	n_CP1_max_speed := GVL_RESD.n_Concrete_Pump_Max_Speed,
	n_CP1_target_speed := UINT_TO_INT(GVL_ROB.in_CP1_set_speed),

	// Admixture pump (High)
	b_AP1_Power_On := GVL_ROB.ib_AP1_power_on,
	b_AP1_Run := GVL_ROB.ib_AP1_set_run,
	b_AP1_Flush_On := GVL_ROB.ib_AP1_flush_on,
	b_AP1_Check_On := GVL_ROB.ib_AP1_check_on,
	
	n_AP1_Flowrate_mode := TRUE,
	n_AP1_Max_Flowrate := UINT_TO_INT(GVL_ROB.on_AP1_max_flowrate),
	n_AP1_Operate_Flowrate := REAL_TO_UDINT((UINT_TO_REAL(GVL_ROB.in_AP1_set_flowrate*10))),
	n_AP1_Check_Flowrate := REAL_TO_UDINT((UINT_TO_REAL(GVL_ROB.in_AP1_set_check_flowrate*10))),
	n_AP1_Flush_Flowrate := REAL_TO_UDINT((UINT_TO_REAL(GVL_ROB.in_AP1_set_flush_flowrate*10))),
	n_AP1_Dosing_factor := UINT_TO_INT(GVL_ROB.in_AP1_set_dosing_factor),
	
	// Admixture pump (High)
	b_SP1_Power_On := GVL_ROB.ib_SP1_power_on,
	b_SP1_Run := GVL_ROB.ib_SP1_set_run,
	b_SP1_Flush_On := GVL_ROB.ib_SP1_flush_on,
	b_SP1_Check_On := GVL_ROB.ib_SP1_set_check_on,
	
	n_SP1_Flowrate_mode := TRUE,
	n_SP1_Max_Flowrate := UINT_TO_INT(GVL_ROB.on_SP1_max_flowrate),
	n_SP1_Operate_Flowrate := REAL_TO_UDINT((UINT_TO_REAL(GVL_ROB.in_SP1_set_flowrate*10))),
	n_SP1_Check_Flowrate := REAL_TO_UDINT((UINT_TO_REAL(GVL_ROB.in_SP1_set_check_flowrate*10))),
	n_SP1_Flush_Flowrate := REAL_TO_UDINT((UINT_TO_REAL(GVL_ROB.in_SP1_flush_flowrate*10))),
	n_SP1_Dosing_factor := UINT_TO_INT(GVL_ROB.in_SP1_dosing_factor),
	);

//***********************************************************************************
// Inline Mixer
//***********************************************************************************
	//mixer 
Mixer1_2(
	Mixer1			:= GVL.Axis_Mixer1,
	Mixer2			:= GVL.Axis_Mixer2,
	f_Velocity		:= GVL.f_MI1_MaxSpeed,
	b_JogForward	:= FALSE,
	b_JogBackwards	:= fb_SetOutputDataToIO.b_MI1_set_run,
	b_Enable		:= fb_SetOutputDataToIO.b_Ml1_Enable AND GVL_IO.ib_CC1_Safety_Ready,
	b_Reset			:= GVL_ROB.ib_CC1_reset OR GVL_IO.ib_CC1_Button_Reset,
	f_Override		:= GVL.n_MI1_OverrideSpeed,
	);
	(*
	fb_MC_SetPosition(
	Axis			:= GVL.Axis_Mixer2,
	memory			:= 1,
	Feedback		:= 0);*)
pos:=GVL.Axis_Mixer2.NcToPlc.ModuloActPos;
GVL.b_MI1_ReadToDrive:=Mixer1_2.b_ReadyToDrive;
P_MI1_OnOff(b_set_run := fb_SetOutputDataToIO.b_MI1_set_run,);

//***********************************************************************************
// Concrete Pump
//***********************************************************************************

// concrete pump power control is from pump itself
P_CP1_Enable();
P_CP1_Check(b_set_run := fb_SetOutputDataToIO.b_CP1_Forward_On,
			b_check_mode_on := fb_SetOutputDataToIO.b_CP1_Check_On,
			t_check_duration := fb_setConfig._t_CP1_Check_Duration,
			);


//***********************************************************************************
// Acceleration Pump
//***********************************************************************************

// Acceleration Pump 1 check
P_AP1_Check(b_set_run := fb_SetOutputDataToIO.b_AP1_Run,
			b_check_mode_on := fb_SetOutputDataToIO.b_AP1_Check_On,
			t_check_duration := fb_setConfig._t_AP1_Check_Duration,
			);
// Check for Acceleration Pump 1 state
IF NOT fb_SetOutputDataToIO.b_AP1_Check_On THEN
//
// Acceleration Pump 1 On/Off
	P_AP1_OnOff(b_set_run := fb_SetOutputDataToIO.b_AP1_Run);
END_IF

//***********************************************************************************
// Superplasticizer Pump
//***********************************************************************************

// Superplasticizer Pump 1 Check (220916 WT
P_SP1_Check(b_set_run := fb_SetOutputDataToIO.b_SP1_Run,
			b_check_mode_on := fb_SetOutputDataToIO.b_SP1_Check_On,
			t_check_duration := fb_setConfig._t_SP1_Check_Duration,
			);
IF NOT fb_SetOutputDataToIO.b_SP1_Check_On THEN
	P_SP1_OnOff(b_set_run := fb_SetOutputDataToIO.b_SP1_Run);
END_IF

//***********************************************************************************
// Get out put data from PLC
//***********************************************************************************
fb_getOutputData(
	
	//CC1
	b_mode_manual := GVL_ROB.ob_mode_manual,
	b_mode_laptop := GVL_ROB.ob_mode_laptop, 	
	b_mode_robot := GVL_ROB.ob_mode_robot, 
	b_CC1_power_on := GVL_ROB.ob_CC1_power_on, 
	n_current_mode := GVL_ROB.on_current_mode,

	//MI1
	b_MI1_Is_Run := GVL_ROB.ob_MI1_is_run,
	b_MI1_is_ready := GVL_ROB.ob_MI1_is_ready,
	n_MI1_status_SpeedM1 := GVL_ROB.on_MI1_status_speed_motor_1,
	n_MI1_status_SpeedM2 := GVL_ROB.on_MI1_status_speed_motor_2,
	f_Status_Torque_Motor_1 := GVL_ROB.on_MI1_status_torque_motor_1,
	f_Status_Torque_Motor_2 := GVL_ROB.on_MI1_status_torque_motor_2,
	f_MI1_status_temperature_funnel_outlet := GVL_ROB.on_MI1_status_temperature_funnel_outlet,
	f_MI1_status_Pressure_funnel_inlet := GVL_ROB.on_MI1_status_pressure_funnel_inlet, 	
	f_MI1_status_temperature_motor_1  := GVL_ROB.on_MI1_status_temperature_motor_1, 			 
	f_MI1_status_temperature_motor_2  := GVL_ROB.on_MI1_status_temperature_motor_2,

	//CP1
	b_CP1_is_run := GVL_ROB.ob_CP1_is_run,
	b_CP1_is_ready := GVL_ROB.ob_CP1_is_ready,
	b_CP1_power_on := GVL_ROB.ob_CP1_power_on,
	b_CP1_safety_grid_on := GVL_ROB.ob_CP1_safety_grid_on,
	b_CP1_drive_error := GVL_ROB.ob_CP1_drive_error,
	
	f_CP1_status_temperature_concrete_fresh := GVL_ROB.on_CP1_status_temperature_concrete_fresh,
	f_CP1_status_temperature_Concrete_pump := GVL_ROB.on_CP1_status_temperature_concrete_pump,
	f_CP1_status_pressure_Concrete_pump := GVL_ROB.on_CP1_status_pressure_concrete_pump,
	
	//AP1
	b_AP1_is_run := GVL_ROB.ob_AP1_is_run,
	b_AP1_is_ready := GVL_ROB.ob_AP1_is_ready,
	b_AP1_no_error := GVL_ROB.ob_AP1_no_error,
	
	//SP1
	b_SP1_is_run := GVL_ROB.ob_SP1_is_run,
	b_SP1_is_ready := GVL_ROB.ob_SP1_is_ready,
	b_SP1_no_error := GVL_ROB.ob_SP1_no_error,
);

END_PROGRAM

// ---- POUs/temp.TcPOU
PROGRAM temp
VAR
END_VAR

(*
// Concrete pump (CP1) *****
	// Digital output from robot (mapping from 16 to 23 in robotstudio )
		arr_CP1_DOSlot := F_CONVERT_BYTE_TO_BIT(GVL_PN.DO_From_ROB[2]);
		GVL_ROB.ib_CP1_forward_on := arr_CP1_DOSlot[0]; // #16
		GVL_ROB.ib_CP1_backward_on := arr_CP1_DOSlot[1];		// 241219 Backward is not working from the conctroller
		GVL_ROB.ib_CP1_check_on := arr_CP1_DOSlot[2];
		GVL_ROB.ib_CP1_flush_on := arr_CP1_DOSlot[3];

	// Group output from Robot ( mapping from 62 to 76, 8*2Bytes in robotstudio)
		F_Convert_2Byte_to_Int(GVL_ROB.in_CP1_set_speed, arr_GOSlot[62], arr_GOSlot[63]); // 0 to 75 [rpm] #62
		F_Convert_2Byte_to_Int(GVL_ROB.in_CP1_set_flowrate, arr_GOSlot[64], arr_GOSlot[65]); // 0 to 16 [l/min]
		F_Convert_2Byte_to_Int(GVL_ROB.in_CP1_set_dosing_volume, arr_GOSlot[66], arr_GOSlot[67]); // calibration in 230926 WT 0.32
		F_Convert_2Byte_to_Int(GVL_ROB.in_CP1_set_check_Flowrate, arr_GOSlot[68], arr_GOSlot[69]);	// [l/min]
		F_Convert_2Byte_to_Int(GVL_ROB.in_CP1_concrete_density, arr_GOSlot[70], arr_GOSlot[71]); // [g/ml]
		F_Convert_2Byte_to_Int(GVL_ROB.in_CP1_concrete_mass, arr_GOSlot[72], arr_GOSlot[73]); // [g]
		F_Convert_2Byte_to_Int(GVL_ROB.in_CP1_set_flush_flowrate, arr_GOSlot[74], arr_GOSlot[75]); // [l/min]
		// F_Convert_2Byte_to_Int(GVL_ROB.t_CP1_set_check_duration, arr_GOSlot[76], arr_GOSlot[77]);	 check with 32 bit


	// Digital input to robot (mapping from 16 to 23 in robotstudio)
		//arr_CP1_DISlot := F_CONVERT_BYTE_TO_BIT(GVL_PN.DI_To_ROB[2]);
		arr_CP1_DISlot[0] := GVL_ROB.ob_CP1_is_run; // #16
		arr_CP1_DISlot[1] := GVL_ROB.ob_CP1_is_ready;

	// Group Input To Robot (mapping from 77 to 91, 8*2Bytes in robotstudio)
		F_Convert_Int_to_2Byte(GVL_ROB.on_CP1_status_temperature_concrete_fresh, arr_GISlot[77], arr_GISlot[78]); // [°C]
		F_Convert_Int_to_2Byte(GVL_ROB.on_CP1_status_temperature_Concrete_pump, arr_GISlot[79], arr_GISlot[80]); // [°C]
		F_Convert_Int_to_2Byte(GVL_ROB.on_CP1_status_pressure_Concrete_pump, arr_GISlot[81], arr_GISlot[82]); // [ bar]




// Admixture pump, High dosage ViscoTech Pump *****
	// Digital output from robot (mapping from 24 to 31 in robotstudio )
		arr_AP1_DOSlot := F_CONVERT_BYTE_TO_BIT(GVL_PN.DO_From_ROB[3]);
		GVL_ROB.ib_AP1_set_run := arr_AP1_DOSlot[0]; // #24
		GVL_ROB.ib_AP1_check_on := arr_AP1_DOSlot[1];
		GVL_ROB.ib_AP1_flush_on := arr_AP1_DOSlot[2];

	// Group output from Robot ( mapping from 77 to 91, 8*2Bytes in robotstudio)
		F_Convert_2Byte_to_Int(GVL_ROB.in_AP1_set_flowrate, arr_GOSlot[77], arr_GOSlot[78]); // **** [ml/min] #77
		F_Convert_2Byte_to_Int(GVL_ROB.in_AP1_set_dosing_factor, arr_GOSlot[79], arr_GOSlot[80]);
		F_Convert_2Byte_to_Int(GVL_ROB.in_AP1_set_check_flowrate, arr_GOSlot[81], arr_GOSlot[82]);
		F_Convert_2Byte_to_Int(GVL_ROB.in_AP1_material_density, arr_GOSlot[83], arr_GOSlot[84]);
		F_Convert_2Byte_to_Int(GVL_ROB.in_AP1_material_mass, arr_GOSlot[85], arr_GOSlot[86]);

		F_Convert_2Byte_to_Int(GVL_ROB.in_AP1_set_dosing_factor, arr_GOSlot[79], arr_GOSlot[80]);
		F_Convert_2Byte_to_Int(GVL_ROB.in_AP1_flush_flowrate, arr_GOSlot[81], arr_GOSlot[82]);
		// F_Convert_2Byte_to_Int(GVL_ROB.t_AP1_set_check_duration, arr_GOSlot[83], arr_GOSlot[84]); check with 32 bit

	// Digital input to robot (mapping from 24 to 31 in robotstudio)
		//arr_AP1_DISlot := F_CONVERT_BYTE_TO_BIT(GVL_PN.DI_To_ROB[3]);	// #24
		arr_AP1_DISlot[0] := GVL_ROB.ob_AP1_is_run;

	// Group Input To Robot (mapping from 92 to 106, 8*2Bytes in robotstudio)
		F_Convert_2Byte_to_Int(GVL_ROB.on_AP1_max_flowrate, arr_GOSlot[92], arr_GOSlot[93]); // [l/min]



// Admixture pump, Low dosage ViscoTech Pump *****
	// Digital output from robot (mapping from 32 to 39 in robotstudio )
		//arr_SP1_DOSlot := F_CONVERT_BYTE_TO_BIT(GVL_PN.DO_From_ROB[4]);
		GVL_ROB.ib_SP1_set_run := arr_SP1_DOSlot[0]; // #32
		GVL_ROB.ib_SP1_set_check_on := arr_SP1_DOSlot[1];
		GVL_ROB.ib_SP1_flush_on := arr_SP1_DOSlot[2];

	// Group output from Robot ( mapping from 92 to 106, 8*2Bytes in robotstudio)
		F_Convert_2Byte_to_Int(GVL_ROB.in_SP1_set_flowrate, arr_GOSlot[92], arr_GOSlot[93]); // **** [ml/min] #92
		F_Convert_2Byte_to_Int(GVL_ROB.in_SP1_dosing_factor, arr_GOSlot[93], arr_GOSlot[94]);
		F_Convert_2Byte_to_Int(GVL_ROB.in_SP1_set_check_flowrate, arr_GOSlot[95], arr_GOSlot[96]);
		F_Convert_2Byte_to_Int(GVL_ROB.in_SP1_material_density, arr_GOSlot[97], arr_GOSlot[98]);
		F_Convert_2Byte_to_Int(GVL_ROB.in_SP1_material_mass, arr_GOSlot[99], arr_GOSlot[100]);
		F_Convert_2Byte_to_Int(GVL_ROB.in_SP1_flush_flowrate, arr_GOSlot[101], arr_GOSlot[102]);
		// F_Convert_2Byte_to_Int(GVL_ROB.t_SP1_Check_Duration, arr_GOSlot[103], arr_GOSlot[104]); // Check with 32 bit

	// Digital input to robot (mapping from 32 to 39 in robotstudio)
		//arr_SP1_DISlot := F_CONVERT_BYTE_TO_BIT(GVL_PN.DI_To_ROB[4]);
		GVL_ROB.ob_SP1_is_run := arr_SP1_DISlot[0]; // #32

	// Group Input To Robot (mapping from 106 to 120, 8*2Bytes in robotstudio)
		F_Convert_2Byte_to_Int(GVL_ROB.on_SP1_max_flowrate, arr_GOSlot[106], arr_GOSlot[107]); // [l/min]>



// Spare Component *****
	// Digital output from robot (mapping from 40 to .. in robotstudio )
		// Template
		// arr_SP1_DOSlot := F_Convert_Byte_to_Bit(GVL_PN.DO_From_ROB[4]);
		// GVL_ROB.ib_SP1_set_run := arr_SP1_DOSlot[0];

	// Group output from Robot ( mapping from 107 to .., 8*2Bytes in robotstudio)
		// F_Convert_2Byte_to_Int(GVL_ROB.in_SP1_set_flowrate, arr_GOSlot[92], arr_GOSlot[93]);
	// Digital input to robot (mapping from 40 to .. in robotstudio)
		// Template
		// arr_SP1_DISlot := F_Convert_Byte_to_Bit(GVL_PN.DI_To_ROB[4]);
		// GVL_ROB.ob_SP1_is_run:= arr_SP1_DISlot[0]; // #32

	// Group Input To Robot (mapping from 121 to .., 8*2Bytes in robotstudio)
		// F_Convert_2Byte_to_Int(GVL_ROB.on_SP1_max_flowrate, arr_GOSlot[106], arr_GOSlot[107]);
//
*)

END_PROGRAM

// ---- POUs/Utils/F_Convert_2Byte_to_Real.TcPOU
FUNCTION F_Convert_2Byte_to_Real

VAR_IN_OUT
	inputNum : REAL; 
	dataByte1 : BYTE;
	dataByte2 : BYTE;
END_VAR

VAR
	arrByte : ARRAY [0..1] OF BYTE;
END_VAR

arrByte[0]:= dataByte1;
arrByte[1]:= dataByte2;
MEMCPY(ADR(inputNum), ADR(arrByte), 2);

//F_Convert_Int_to_2Byte:=arrByte;

END_FUNCTION

// ---- POUs/Utils/F_Convert_Bit_to_Byte.TcPOU
FUNCTION  F_Convert_Bit_to_Byte
VAR_IN_OUT
	//dataByte : BYTE;
	arrBool : ARRAY[0..7] OF BOOL;
	dataByte : BYTE;
END_VAR

VAR
	i : INT; 
	arrBool_temp : ARRAY[0..7] OF BOOL;
END_VAR

// ***********************************************************************************
//
// Müller-steinag Gruppe, Kandergrien Einigen, CH-3646 Bern
// ETH Zurich, Building HIF E26, Laura-Hezner-Weg 7, CH-8093 Zürich
// 
// ***********************************************************************************
// 
// PROJECT     :  A061 Digital Casting System 
// FUNCTION    :  Data Converter Bit to Byte
// AUTHOR      :  Weiting Chen
// EMAIL       :  chenw@usi.ch
// Copyright   :  USI Mendrisio; ETH Zürich; Müller-steinag Gruppe (CH) 2023
//
// ***********************************************************************************


//MEMCPY(ADR(dataByte), ADR(arrBool), SIZEOF(arrBool));
arrBool_temp[0] := BYTE_TO_BIT(dataByte AND 16#1);
arrBool_temp[1] := BYTE_TO_BIT(dataByte AND 16#2);
arrBool_temp[2] := BYTE_TO_BIT(dataByte AND 16#4);
arrBool_temp[3] := BYTE_TO_BIT(dataByte AND 16#8);
arrBool_temp[4] := BYTE_TO_BIT(dataByte AND 16#10);
arrBool_temp[5] := BYTE_TO_BIT(dataByte AND 16#20);
arrBool_temp[6] := BYTE_TO_BIT(dataByte AND 16#40);
arrBool_temp[7] := BYTE_TO_BIT(dataByte AND 16#80);


arrBool_temp[0] := arrBool[0];
arrBool_temp[1] := arrBool[1];
arrBool_temp[2] := arrBool[2];
arrBool_temp[3] := arrBool[3];
arrBool_temp[4] := arrBool[4];
arrBool_temp[5] := arrBool[5];
arrBool_temp[6] := arrBool[6];
arrBool_temp[7] := arrBool[7];

END_FUNCTION
